// TIA Portal V20 export
DATA_BLOCK "CallUnit_DB"   // DB147
// stored: AssignedProDiagFB Unit1.ProDiag, InstanceOfName Unit1.CallUnit, InstanceOfType FB, Namespace Unit1
"Unit1.CallUnit"
   // VAR_INPUT
   //    safetyReleased : Bool;
   // END_VAR
   // VAR_OUTPUT
   //    acknowledgeSafety { ExternalWritable := 'False'} : Bool;
   // END_VAR
   // VAR_IN_OUT
   //    globalStatus : "LAF_typeGeneralStatus";
   //    unitInterface : "LAF_typeUnitInterface";
   // END_VAR
   // VAR
   //    instManageAlarms { ExternalWritable := 'False'} : "LAF_ManageAlarms";
   //    instStatusCollector { ExternalWritable := 'False'} : "LUC_StatusCollector";
   //    instInterfaceManager { ExternalWritable := 'False'} : "LUC_InterfaceManager";
   //    instUnitModeStateManager { ExternalWritable := 'False'} : "LPMLV2022_UnitModeStateManager";
   //    instRemoteInterfaceOpcUa { ExternalWritable := 'False'} : "LUC_RemoteCtrl_OpcUa";
   //    instSignalStack { ExternalWritable := 'False'} : "LUC_SignalStack";
   //    instUnitModeStateTimes { ExternalWritable := 'False'} : "LPMLV2022_UnitModeStateTimes";
   //    instUnitModeChangeAllowed { ExternalWritable := 'False'} : "LPMLV2022_UnitModeChangeAllowed";
   //    instPFEEvents { ExternalWritable := 'False'} : "Unit1.EventsPFE";
   //    instEQP_Interface_BA030 { ExternalWritable := 'False'} : "LER_EQP_Interface";
   //    instEQP_Interface_BA040 { ExternalWritable := 'False'} : "LER_EQP_Interface";
   //    instEQP_Interface_BA100 { S7_SetPoint := 'True'} : "LER_EQP_m_Interface";
   //    instEQP_Interface_CoveyorA { ExternalWritable := 'False'} : "LER_EQP_Communication";
   //    instSinaInfeed { ExternalWritable := 'False'} : SinaInfeed;
   //    statRemoteInterface { ExternalWritable := 'False'} : "LUC_typeCommands";
   //    statLocalInterface { ExternalWritable := 'False'} : "LUC_typeCommands";
   //    statEmEnableCheck { ExternalWritable := 'False'} : Array[0..2] of Bool;
   //    statEmHomeScCheck { ExternalWritable := 'False'} : Array[0..9] of Bool;
   //    statRunOutStatusCheck { ExternalWritable := 'False'} : Array[0..9] of Bool;
   //    statEOCStatusCheck { ExternalWritable := 'False'} : Array[0..19] of Bool;
   //    statPartData { ExternalWritable := 'False'} : Struct
   //       BA030 : "LER_typePartData";
   //       BA040 : "LER_typePartData";
   //    END_STRUCT;
   //    statDataDelete { ExternalWritable := 'False'} : "LER_typePartData";
   //    statTonTime { ExternalWritable := 'False'} : Array[0..99] of TON_TIME;
   //    statTofTime { ExternalWritable := 'False'} : Array[0..9] of TOF_TIME;
   //    statFlipFlop { ExternalWritable := 'False'} : Array[0..99] of Bool;
   //    statPulse { ExternalWritable := 'False'} : Array[0..9999] of Bool;
   //    statNoModeCmd { ExternalWritable := 'False'} : Bool;
   //    statEnableManualCmds { ExternalWritable := 'False'} : Bool;
   //    InstLER_FFU_LIU117 { S7_SetPoint := 'True'} : "LER_FFU_LIU117";
   //    ClearData { S7_SetPoint := 'True'} : "LER_typePartData";
   //    Data_TrCondition { S7_SetPoint := 'True'} : Array[0..20] of Bool;
   //    NoData_Alarm : Array[0..20] of Bool;
   //    statAllEmLinked : Bool;
   //    citi_Ptrig : Array[0..20] of Bool;
   //    citiTon : Array[0..20] of TON_TIME;
   //    citi : Time;
   //    citiTest : Array[0..20] of Bool;
   //    instMQTTClient { S7_SetPoint := 'True'} : "LMQTT_Client";
   //    instPFEUnit { S7_SetPoint := 'True'} : "Unit1.EventsPFE_Unit";
   // END_VAR
BEGIN
END_DATA_BLOCK
